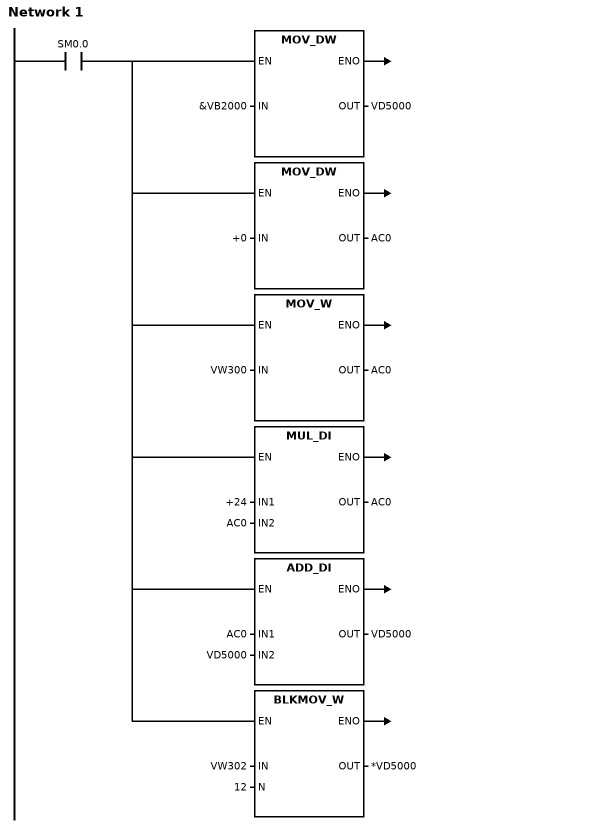
[picture p48: SBR5 networks 1-1]
Network 1
LD     SM0.0
MOVD   &VB2000, VD5000
MOVD   +0, AC0
MOVW   VW300, AC0
*D     +24, AC0
+D     AC0, VD5000
BMW    VW302, *VD5000, 12
END_SUBROUTINE_BLOCK

SUBROUTINE_BLOCK 读工艺:SBR6
TITLE=
BEGIN
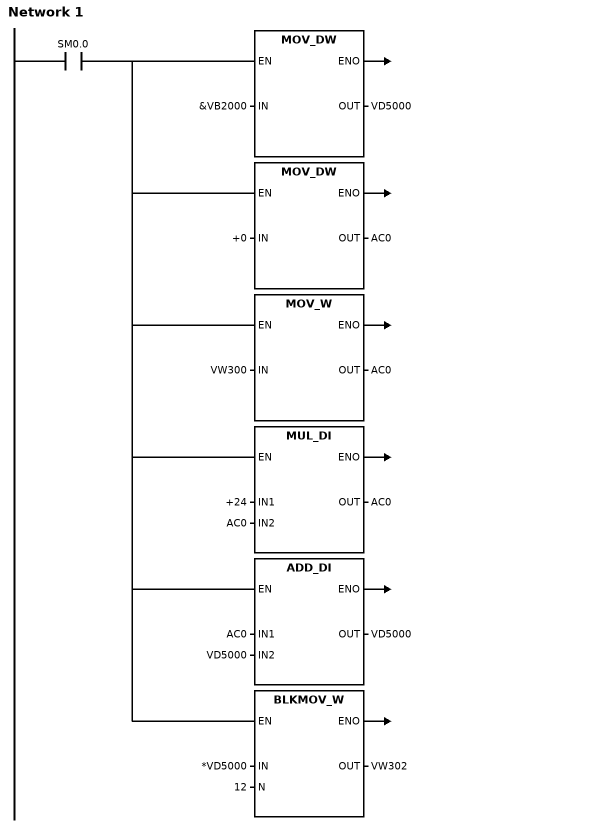
Network 1
LD     SM0.0
MOVD   &VB2000, VD5000
MOVD   +0, AC0
MOVW   VW300, AC0
*D     +24, AC0
+D     AC0, VD5000
BMW    *VD5000, VW302, 12
END_SUBROUTINE_BLOCK

SUBROUTINE_BLOCK 存EEPROM:SBR7
TITLE=
BEGIN
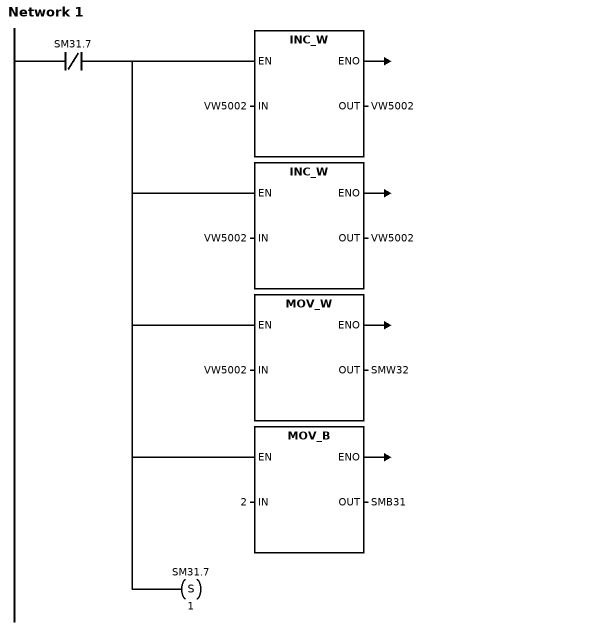
Network 1
LDN    SM31.7
INCW   VW5002
INCW   VW5002
MOVW   VW5002, SMW32
MOVB   2, SMB31
S      SM31.7, 1
END_SUBROUTINE_BLOCK

SUBROUTINE_BLOCK 分合设置:SBR9
TITLE=
BEGIN
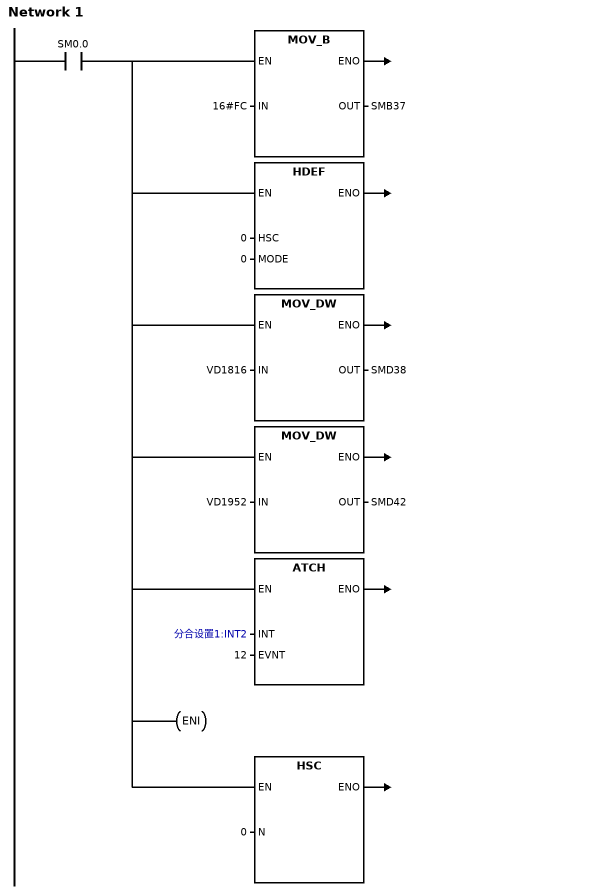
Network 1
LD     SM0.0
MOVB   16#FC, SMB37
HDEF   0, 0
MOVD   VD1816, SMD38
MOVD   VD1952, SMD42
ATCH   分合设置1:INT2, 12
ENI
HSC    0
END_SUBROUTINE_BLOCK

SUBROUTINE_BLOCK 全机运行频率计算:SBR10
TITLE=
BEGIN
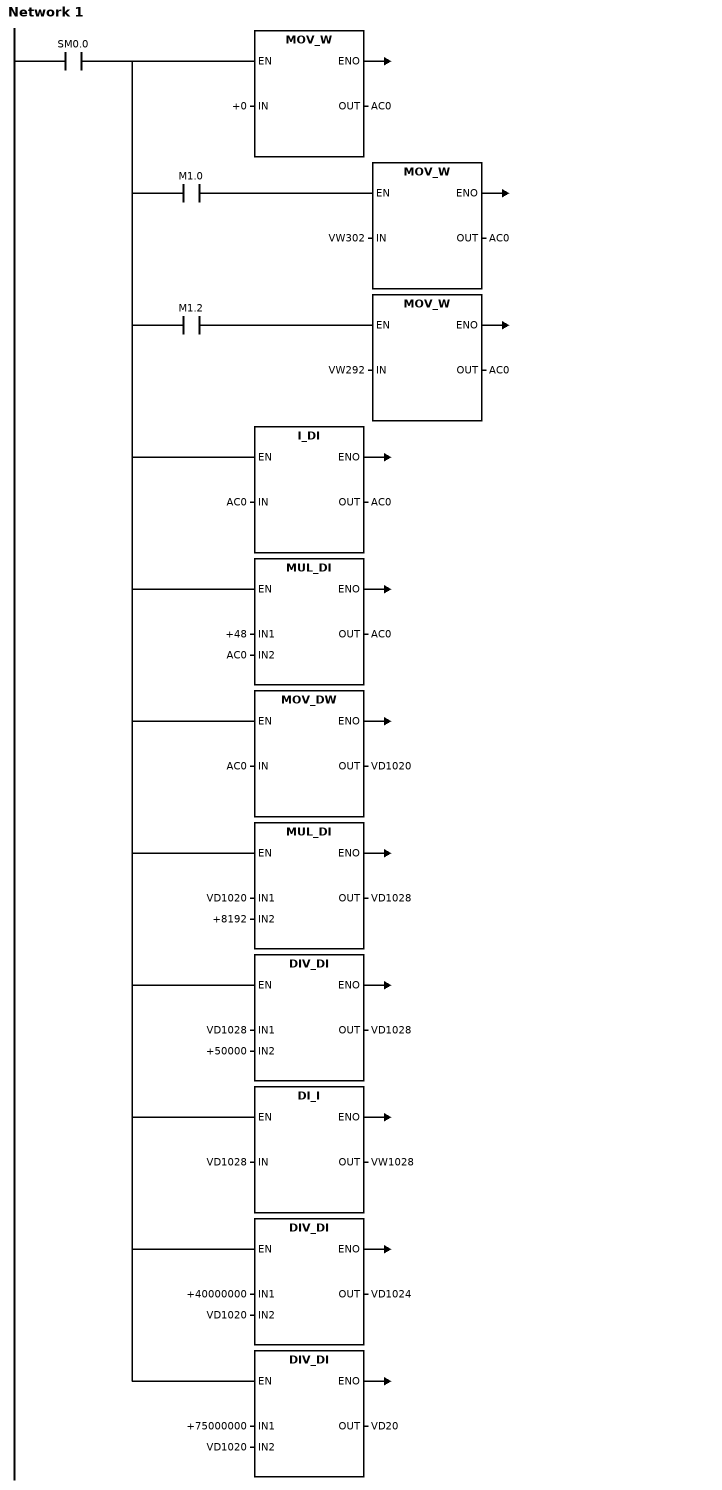
Network 1
LD     SM0.0
LPS
MOVW   +0, AC0
A      M1.0
MOVW   VW302, AC0
LRD
A      M1.2
MOVW   VW292, AC0
LRD
ITD    AC0, AC0
LRD
*D     +48, AC0
LRD
MOVD   AC0, VD1020
LRD
MOVD   VD1020, VD1028
*D     +8192, VD1028
LRD
/D     +50000, VD1028
LRD
DTI    VD1028, VW1028
LRD
MOVD   +40000000, VD1024
/D     VD1020, VD1024
LPP
MOVD   +75000000, VD20
/D     VD1020, VD20
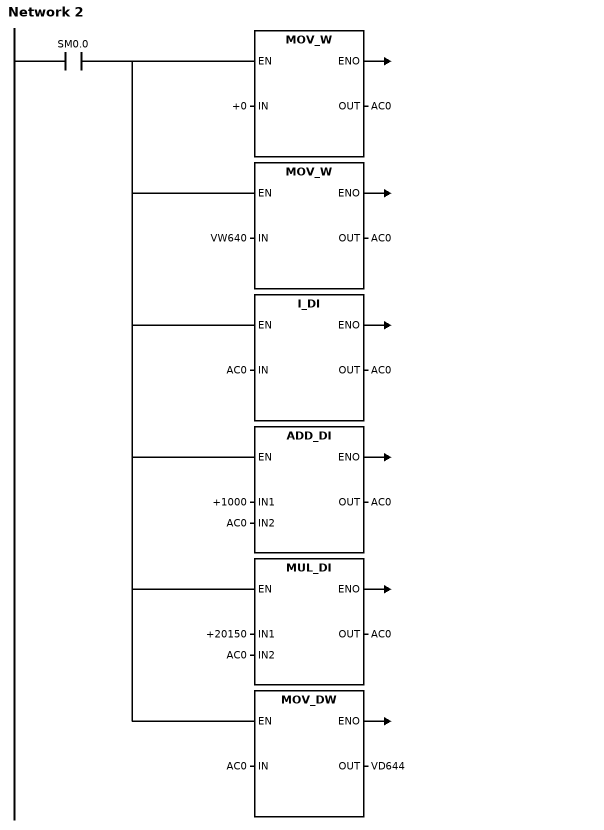
Network 2
LD     SM0.0
MOVW   +0, AC0
MOVW   VW640, AC0
ITD    AC0, AC0
+D     +1000, AC0
*D     +20150, AC0
MOVD   AC0, VD644
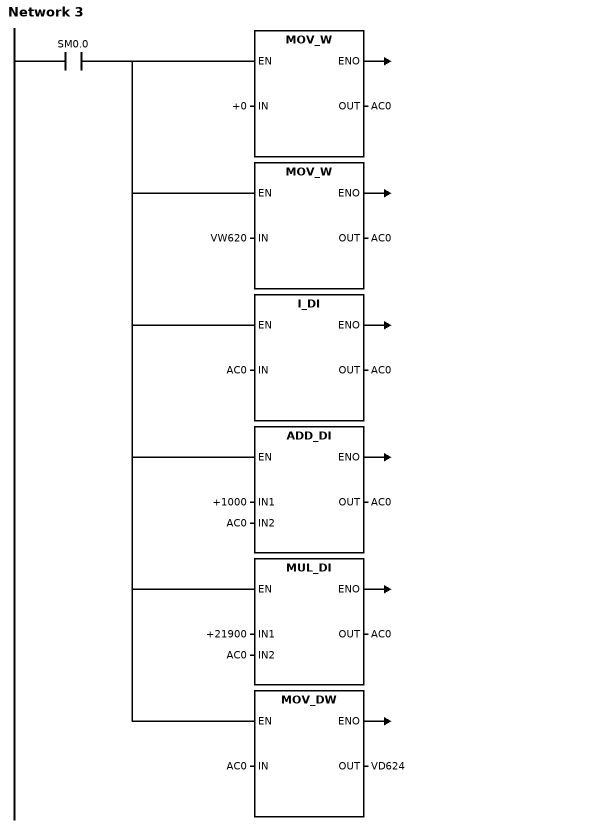
Network 3
LD     SM0.0
MOVW   +0, AC0
MOVW   VW620, AC0
ITD    AC0, AC0
+D     +1000, AC0
*D     +21900, AC0
MOVD   AC0, VD624
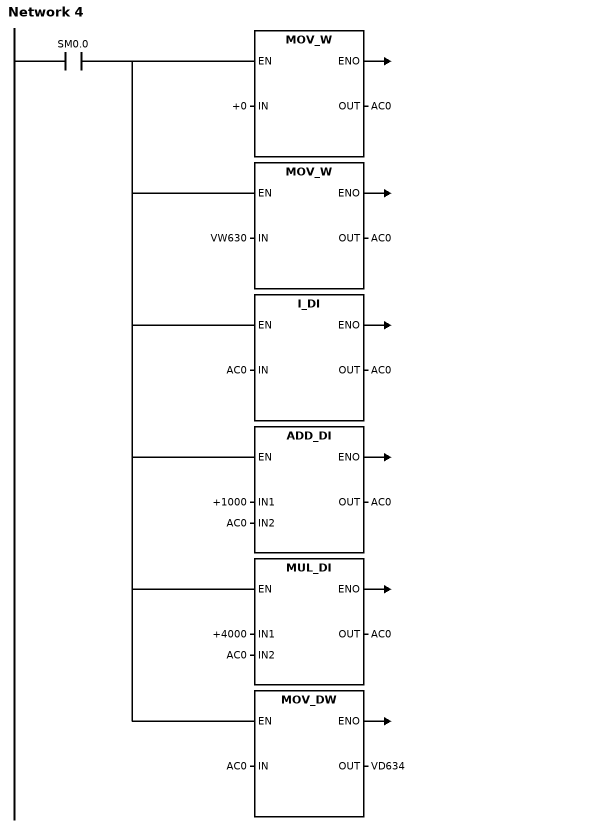
Network 4
LD     SM0.0
MOVW   +0, AC0
MOVW   VW630, AC0
ITD    AC0, AC0
+D     +1000, AC0
*D     +4000, AC0
MOVD   AC0, VD634
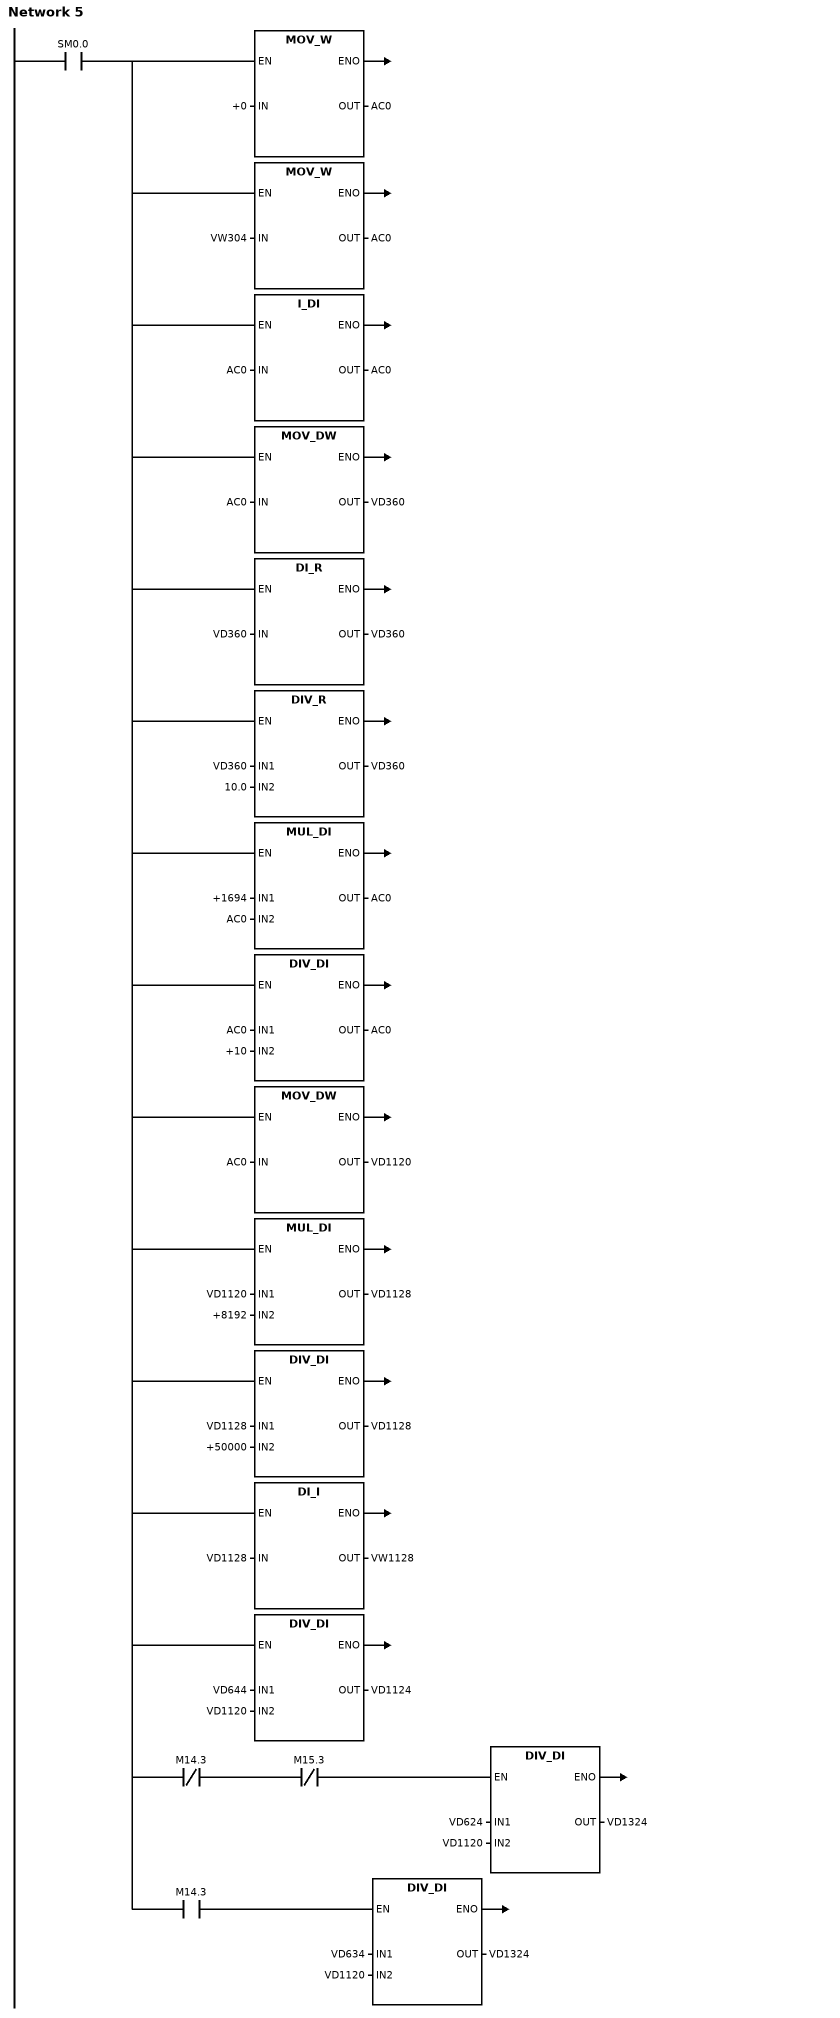
Network 5
LD     SM0.0
LPS
MOVW   +0, AC0
MOVW   VW304, AC0
ITD    AC0, AC0
MOVD   AC0, VD360
DTR    VD360, VD360
/R     10.0, VD360
*D     +1694, AC0
/D     +10, AC0
MOVD   AC0, VD1120
MOVD   VD1120, VD1128
*D     +8192, VD1128
/D     +50000, VD1128
DTI    VD1128, VW1128
MOVD   VD644, VD1124
/D     VD1120, VD1124
AN     M14.3
AN     M15.3
MOVD   VD624, VD1324
/D     VD1120, VD1324
LPP
A      M14.3
MOVD   VD634, VD1324
/D     VD1120, VD1324
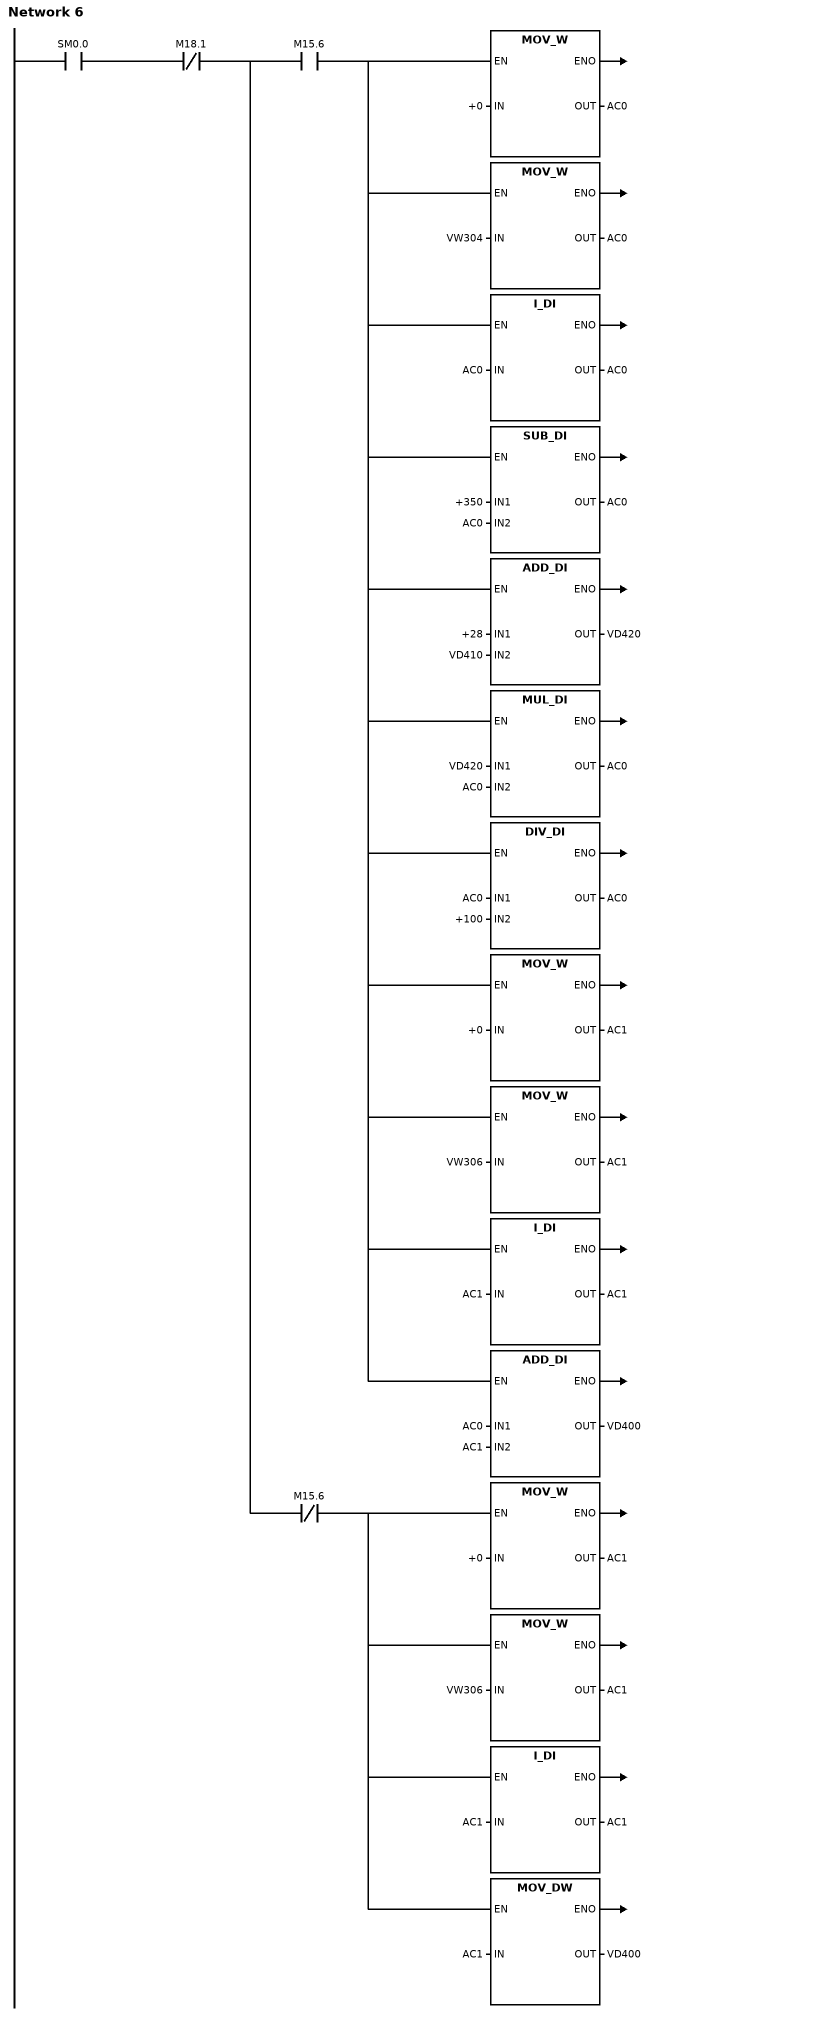
Network 6
LD     SM0.0
AN     M18.1
LPS
A      M15.6
MOVW   +0, AC0
MOVW   VW304, AC0
ITD    AC0, AC0
INVD   AC0
INCD   AC0
+D     +350, AC0
MOVD   +28, VD420
+D     VD410, VD420
*D     VD420, AC0
/D     +100, AC0
MOVW   +0, AC1
MOVW   VW306, AC1
ITD    AC1, AC1
MOVD   AC0, VD400
+D     AC1, VD400
LPP
AN     M15.6
MOVW   +0, AC1
MOVW   VW306, AC1
ITD    AC1, AC1
MOVD   AC1, VD400
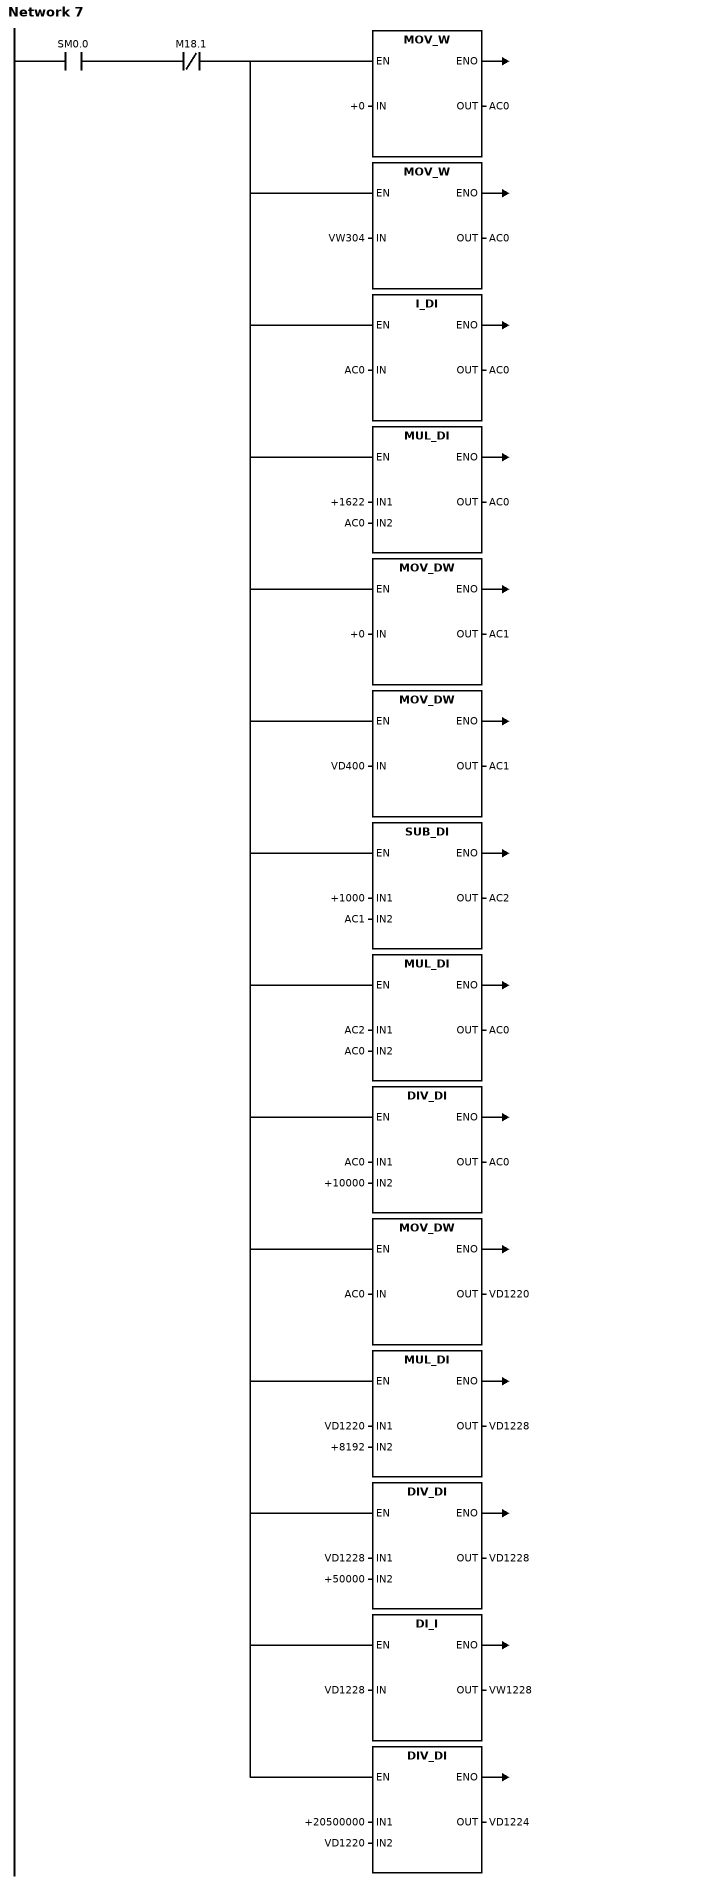
Network 7
LD     SM0.0
AN     M18.1
MOVW   +0, AC0
MOVW   VW304, AC0
ITD    AC0, AC0
*D     +1622, AC0
MOVD   +0, AC1
MOVD   VD400, AC1
MOVD   +1000, AC2
-D     AC1, AC2
*D     AC2, AC0
/D     +10000, AC0
MOVD   AC0, VD1220
MOVD   VD1220, VD1228
*D     +8192, VD1228
/D     +50000, VD1228
DTI    VD1228, VW1228
MOVD   +20500000, VD1224
/D     VD1220, VD1224
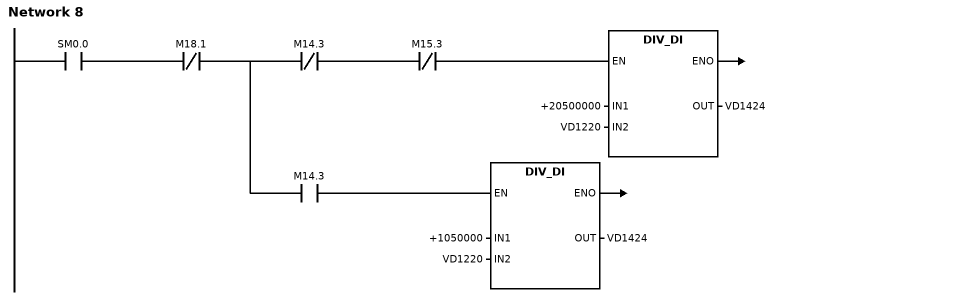
Network 8
LD     SM0.0
AN     M18.1
LPS
AN     M14.3
AN     M15.3
MOVD   +20500000, VD1424
/D     VD1220, VD1424
LPP
A      M14.3
MOVD   +1050000, VD1424
/D     VD1220, VD1424
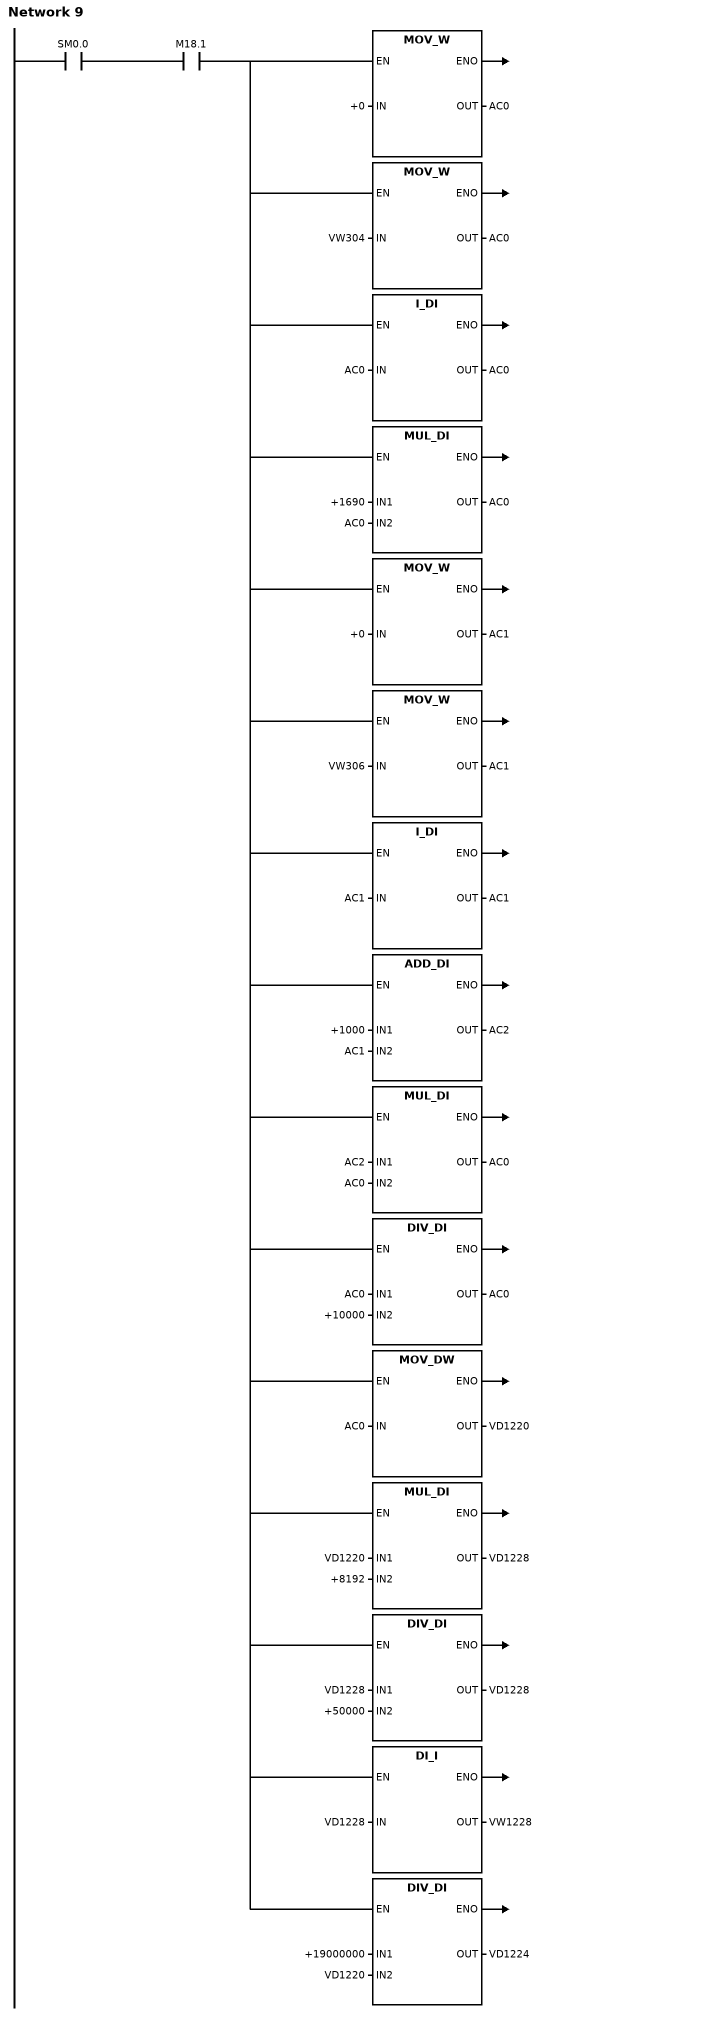
Network 9
LD     SM0.0
A      M18.1
MOVW   +0, AC0
MOVW   VW304, AC0
ITD    AC0, AC0
*D     +1690, AC0
MOVW   +0, AC1
MOVW   VW306, AC1
ITD    AC1, AC1
MOVD   +1000, AC2
+D     AC1, AC2
*D     AC2, AC0
/D     +10000, AC0
MOVD   AC0, VD1220
MOVD   VD1220, VD1228
*D     +8192, VD1228
/D     +50000, VD1228
DTI    VD1228, VW1228
MOVD   +19000000, VD1224
/D     VD1220, VD1224
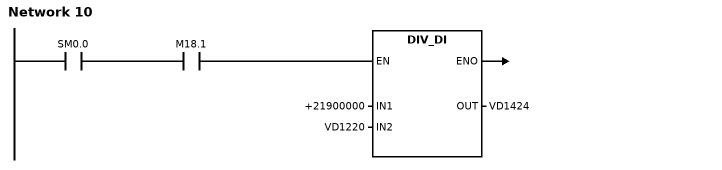
Network 10
LD     SM0.0
A      M18.1
MOVD   +21900000, VD1424
/D     VD1220, VD1424
END_SUBROUTINE_BLOCK

SUBROUTINE_BLOCK 部分运行频率计算:SBR11
TITLE=
BEGIN
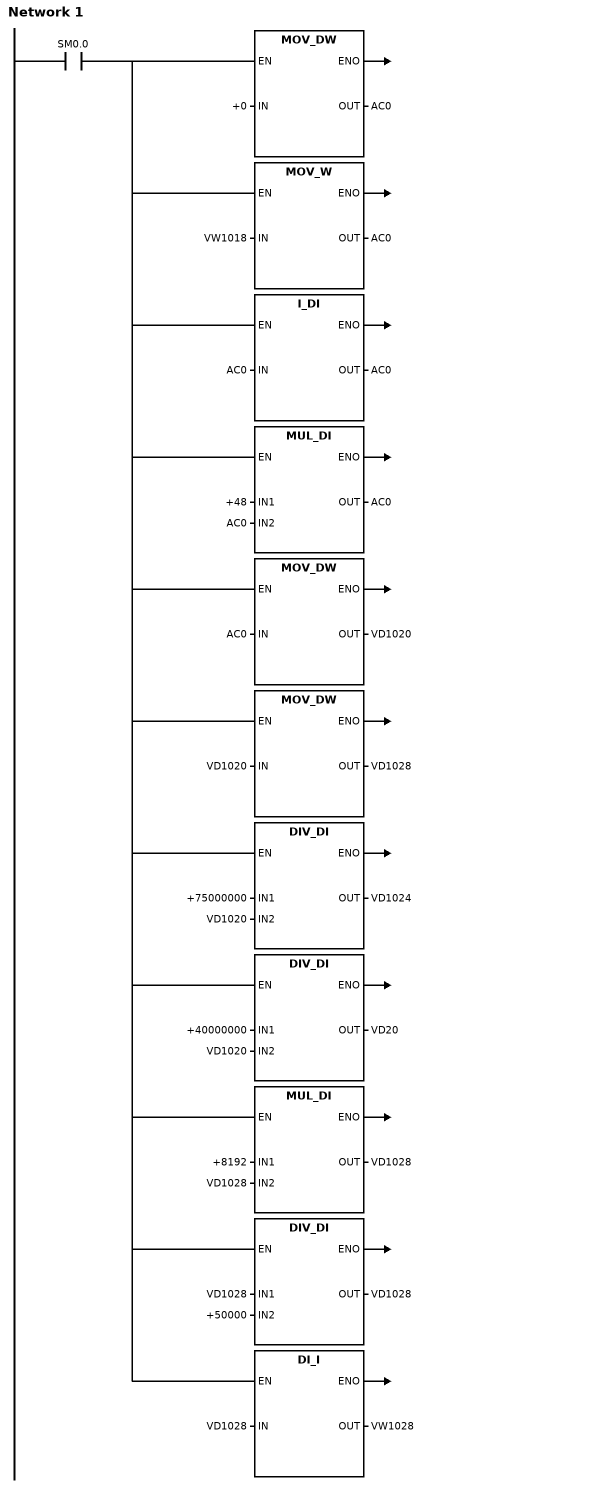
Network 1
LD     SM0.0
MOVD   +0, AC0
MOVW   VW1018, AC0
ITD    AC0, AC0
*D     +48, AC0
MOVD   AC0, VD1020
MOVD   VD1020, VD1028
MOVD   +75000000, VD1024
/D     VD1020, VD1024
MOVD   +40000000, VD20
/D     VD1020, VD20
*D     +8192, VD1028
/D     +50000, VD1028
DTI    VD1028, VW1028
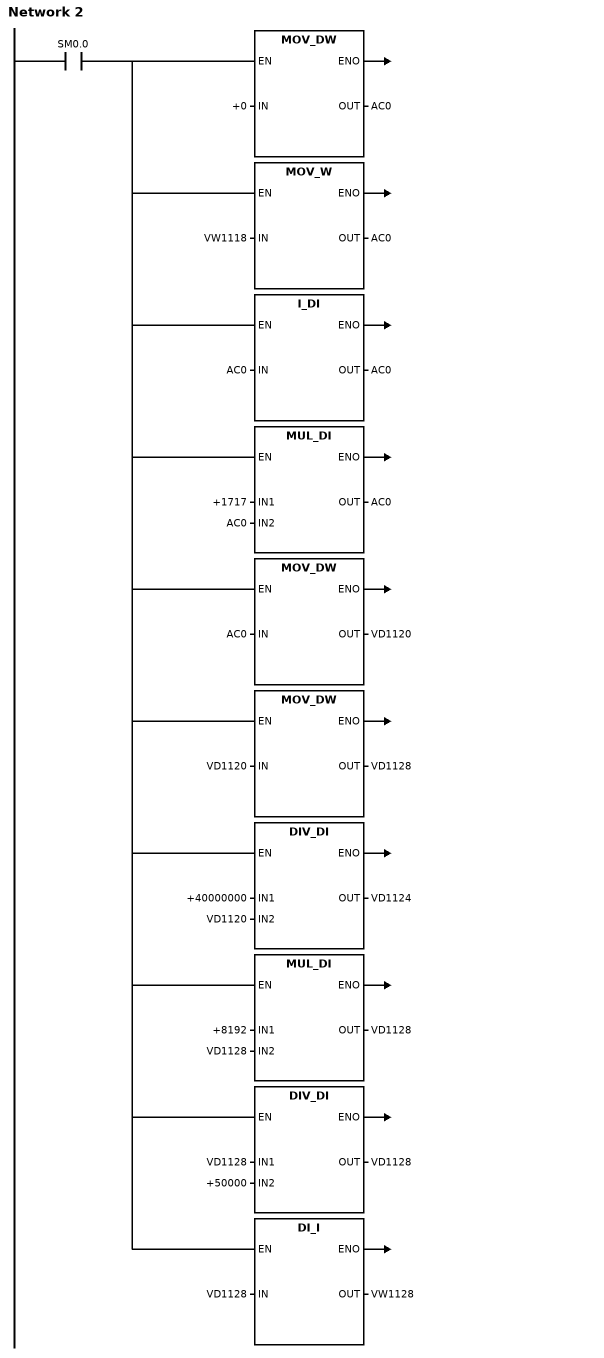
Network 2
LD     SM0.0
MOVD   +0, AC0
MOVW   VW1118, AC0
ITD    AC0, AC0
*D     +1717, AC0
MOVD   AC0, VD1120
MOVD   VD1120, VD1128
MOVD   +40000000, VD1124
/D     VD1120, VD1124
*D     +8192, VD1128
/D     +50000, VD1128
DTI    VD1128, VW1128
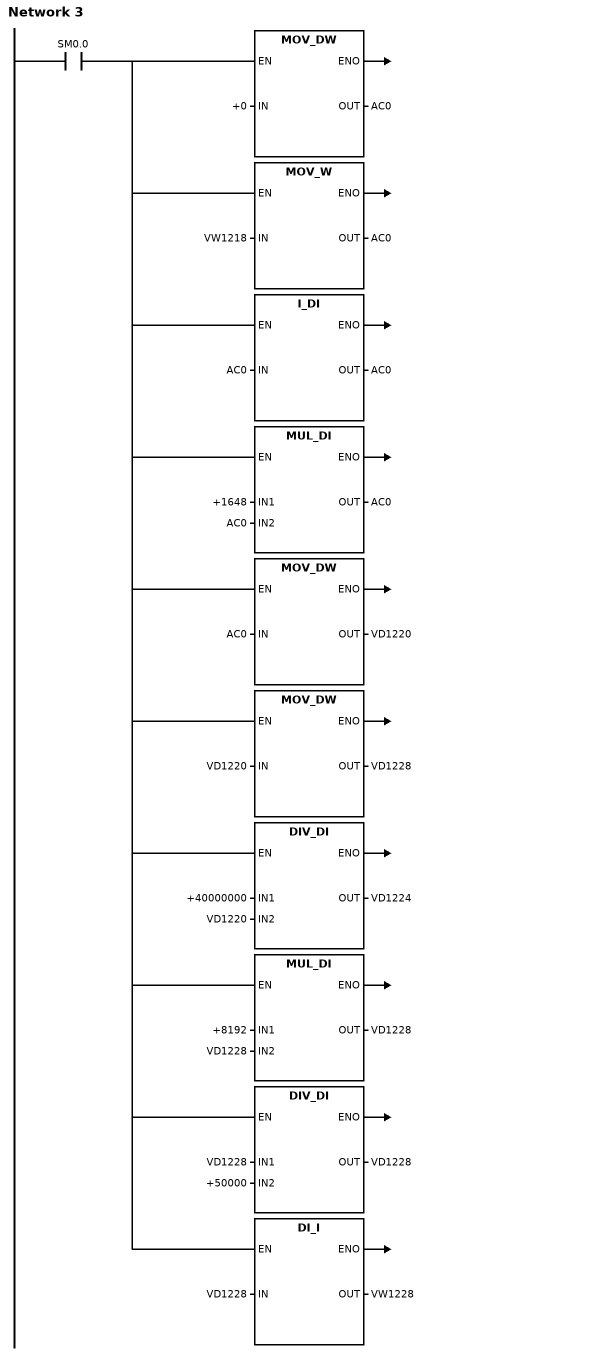
Network 3
LD     SM0.0
MOVD   +0, AC0
MOVW   VW1218, AC0
ITD    AC0, AC0
*D     +1648, AC0
MOVD   AC0, VD1220
MOVD   VD1220, VD1228
MOVD   +40000000, VD1224
/D     VD1220, VD1224
*D     +8192, VD1228
/D     +50000, VD1228
DTI    VD1228, VW1228
END_SUBROUTINE_BLOCK

SUBROUTINE_BLOCK 送公共参数:SBR13
TITLE=
BEGIN
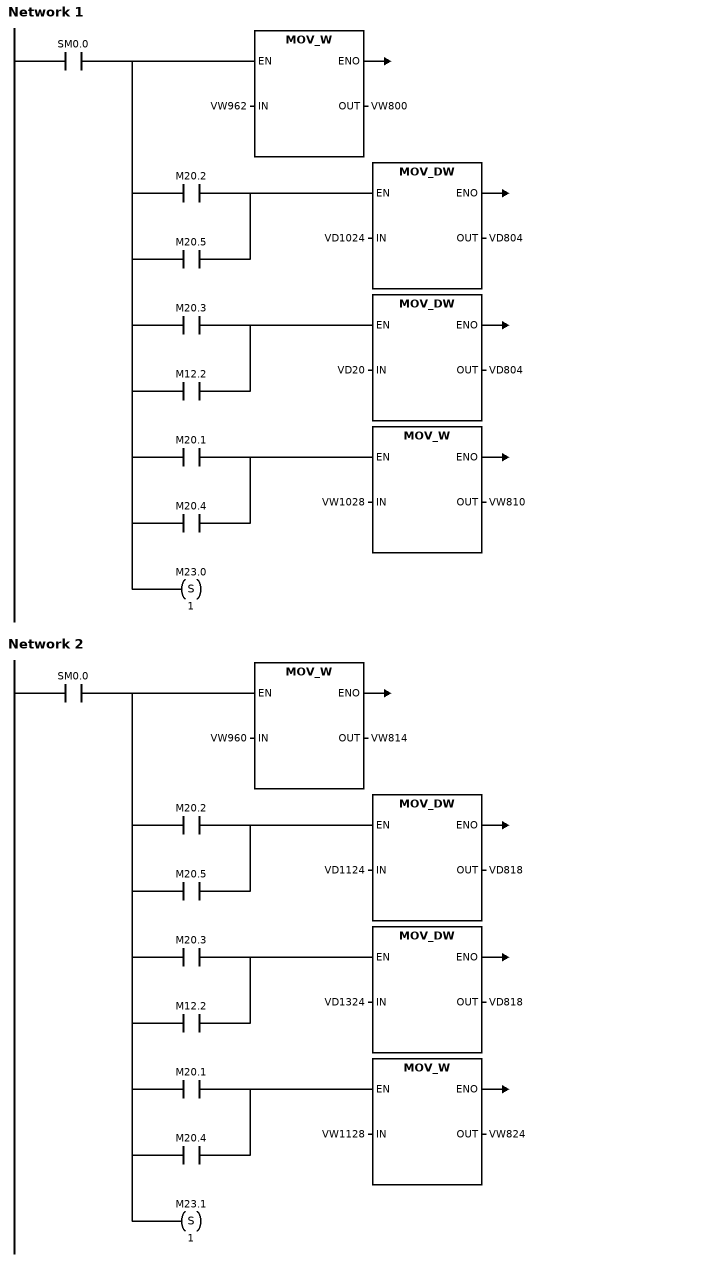
Network 1
LD     SM0.0
LPS
MOVW   VW962, VW800
LD     M20.2
O      M20.5
ALD
MOVD   VD1024, VD804
LRD
LD     M20.3
O      M12.2
ALD
MOVD   VD20, VD804
LRD
LD     M20.1
O      M20.4
ALD
MOVW   VW1028, VW810
LPP
S      M23.0, 1
Network 2
LD     SM0.0
LPS
MOVW   VW960, VW814
LD     M20.2
O      M20.5
ALD
MOVD   VD1124, VD818
LRD
LD     M20.3
O      M12.2
ALD
MOVD   VD1324, VD818
LRD
LD     M20.1
O      M20.4
ALD
MOVW   VW1128, VW824
LPP
S      M23.1, 1
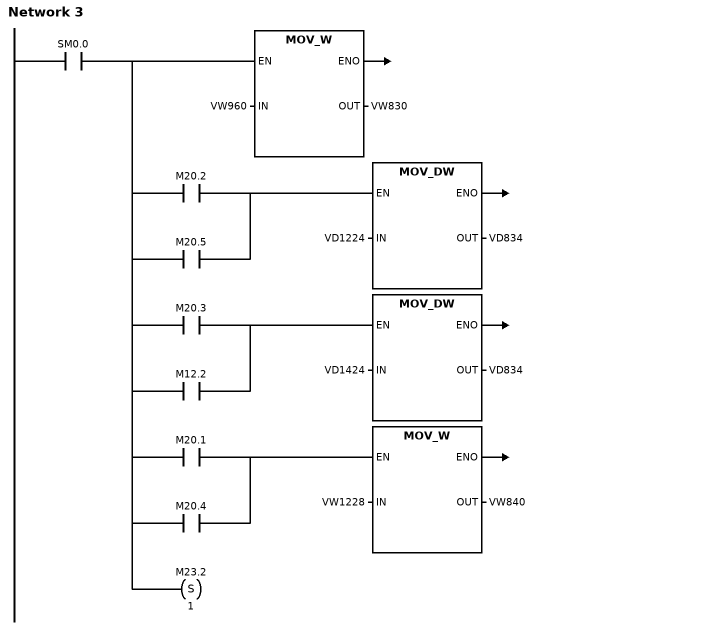
Network 3
LD     SM0.0
LPS
MOVW   VW960, VW830
LD     M20.2
O      M20.5
ALD
MOVD   VD1224, VD834
LRD
LD     M20.3
O      M12.2
ALD
MOVD   VD1424, VD834
LRD
LD     M20.1
O      M20.4
ALD
MOVW   VW1228, VW840
LPP
S      M23.2, 1
END_SUBROUTINE_BLOCK

SUBROUTINE_BLOCK 变频器控制:SBR16
TITLE=
BEGIN
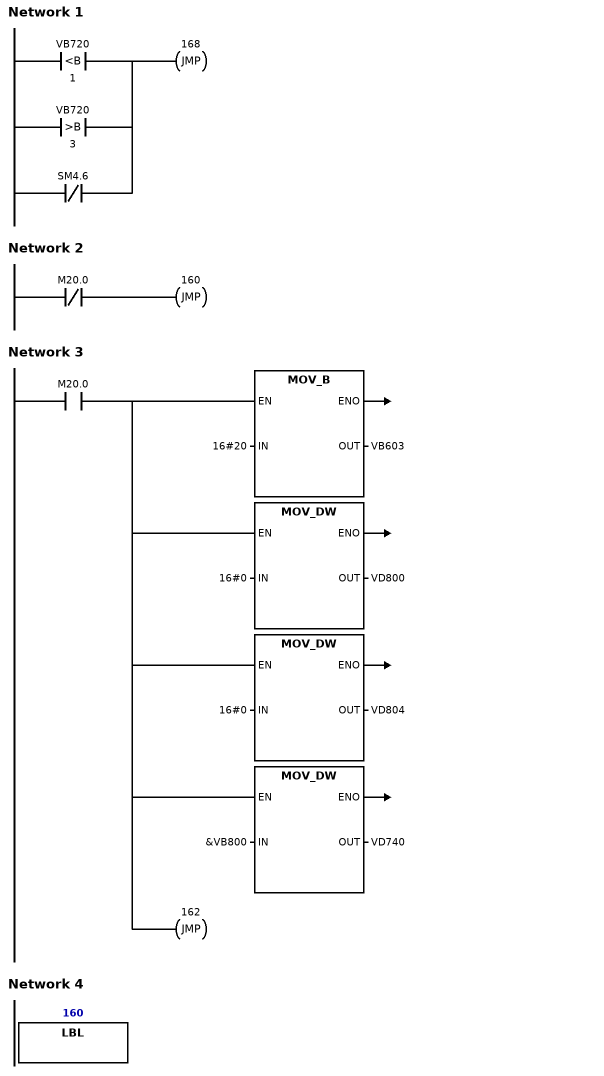
Network 1
LDB<   VB720, 1
OB>    VB720, 3
ON     SM4.6
JMP    168
Network 2
LDN    M20.0
JMP    160
Network 3
LD     M20.0
MOVB   16#20, VB603
MOVD   16#0, VD800
MOVD   16#0, VD804
MOVD   &VB800, VD740
JMP    162
Network 4
LBL    160
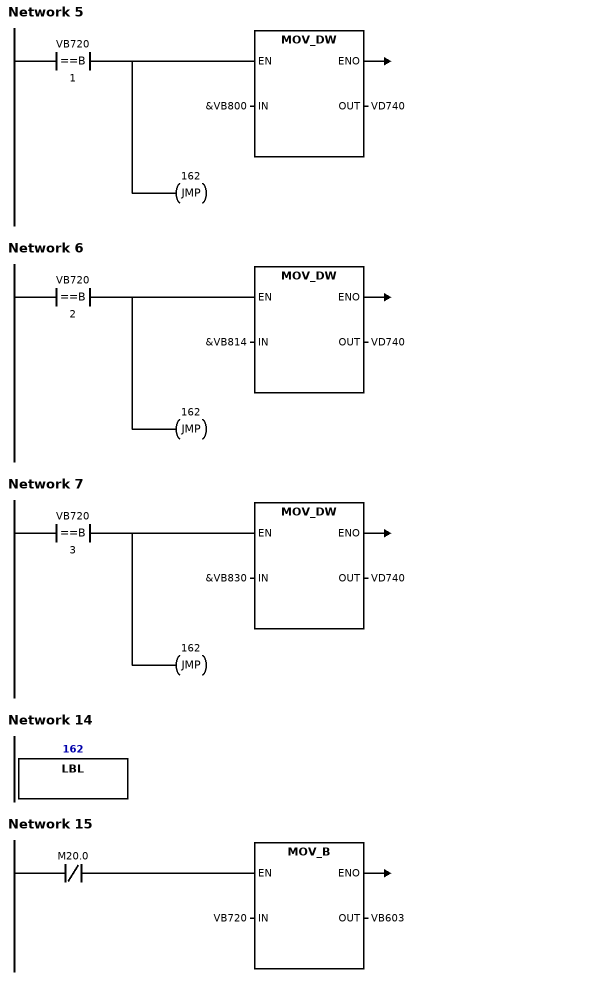
Network 5
LDB=   VB720, 1
MOVD   &VB800, VD740
JMP    162
Network 6
LDB=   VB720, 2
MOVD   &VB814, VD740
JMP    162
Network 7
LDB=   VB720, 3
MOVD   &VB830, VD740
JMP    162
Network 14
LBL    162
Network 15
LDN    M20.0
MOVB   VB720, VB603
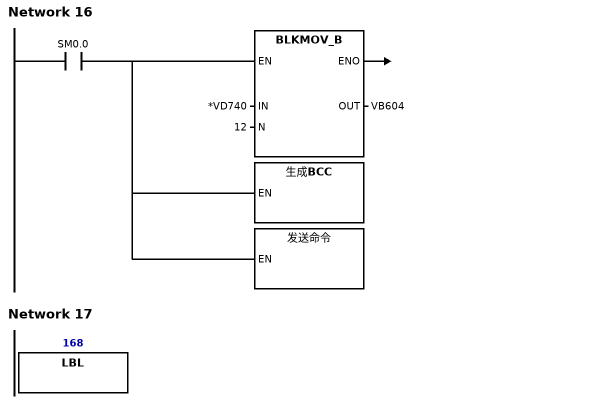
Network 16
LD     SM0.0
BMB    *VD740, VB604, 12
CALL   生成BCC:SBR2
CALL   发送命令:SBR1
Network 17
LBL    168
END_SUBROUTINE_BLOCK

INTERRUPT_BLOCK 发送完成:INT0
TITLE=中断程序注释
BEGIN
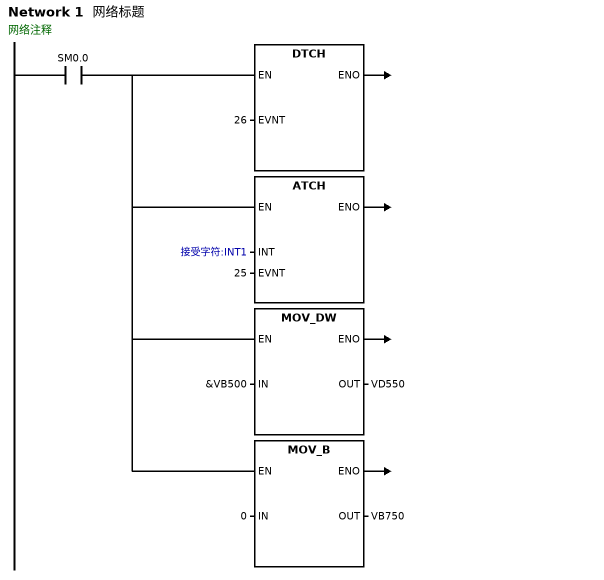
Network 1 // 网络标题
// 网络注释
LD     SM0.0
DTCH   26
ATCH   接受字符:INT1, 25
MOVD   &VB500, VD550
MOVB   0, VB750
END_INTERRUPT_BLOCK

INTERRUPT_BLOCK 接受字符:INT1
TITLE=
BEGIN
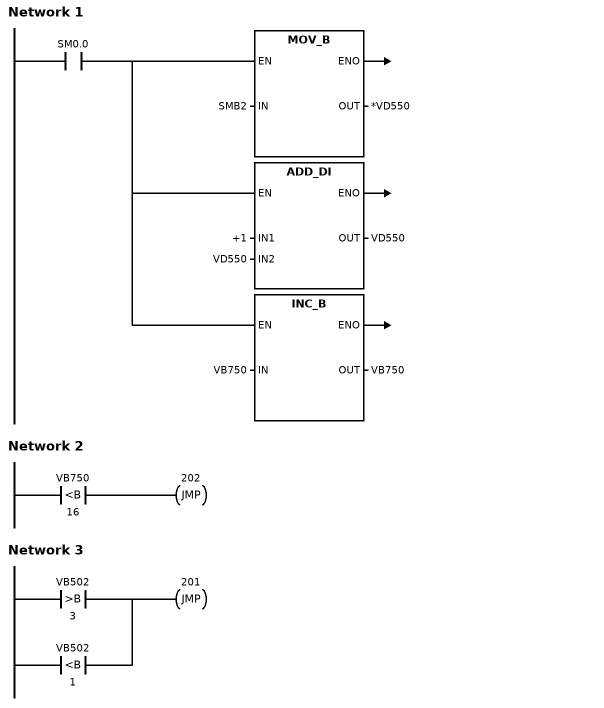
Network 1
LD     SM0.0
MOVB   SMB2, *VD550
+D     +1, VD550
INCB   VB750
Network 2
LDB<   VB750, 16
JMP    202
Network 3
LDB>   VB502, 3
OB<    VB502, 1
JMP    201
